(* CODESYS project FU_dwBitSet.xml

Project tree, tasks and I/O mapping:
  function FU_dwBitSet [ST]
*)

// FU_dwBitSet
//This function sets the bit value from a variable
// |**Version**|**Author**| **Date** |**Changes**
// | 1         | NSN      | 11-01-19 | Creation
FUNCTION FU_dwBitSet : BOOL
VAR_IN_OUT
	dbVar	:DWORD;		//The value to work with
END_VAR
VAR_INPUT
	bIndex		:BYTE;		//Which bit to get
	xVal		:BOOL;		//What to set the bit to
END_VAR

dbVar		:=		(dbVar AND NOT(SHL(TO_DWORD(1),bIndex))) OR (SHL(TO_DWORD(xVal),bIndex));

END_FUNCTION
